PROGRAM TelescopeAuxiliary
VAR
	MQTTTimer : TON := (PT:=T#5S);
END_VAR
VAR_INPUT
	comm: I_Comm;
END_VAR
VAR_OUTPUT
	// BT9 mirror
	temperature_mirror2:	REAL;
	// BT10
	temperature_mirror1:	REAL;
END_VAR

temperature_mirror1 := GVL_Telescope.temperature_mirror1 / 1000.0;
temperature_mirror2 := GVL_Telescope.temperature_mirror2 / 1000.0;

MQTTTimer(IN:=TRUE);
IF MQTTTimer.Q THEN // publish new payload every second

	comm.Publish('telescope', 'dome', 'Mirror1Temperature',	LREAL_TO_FMTSTR(temperature_mirror1, 2, TRUE));
	comm.Publish('telescope', 'dome', 'Mirror2Temperature',	LREAL_TO_FMTSTR(temperature_mirror2, 2, TRUE));
	
	MQTTTimer(IN:=FALSE);

END_IF

END_PROGRAM

(* stored: Version 1.1.0.1, ProductVersion 3.1.4026.8
   POU TelescopeAuxiliary: Id {974ce34a-6026-4bc5-b92d-99da70a09948}, SpecialFunc None *)
